{attribute 'qualified_only'}
VAR_GLOBAL

	Par1 		:BOOL:=TRUE;
	Par2		:INT:=10;
	Par3		:DINT:=100;
	Par4		:REAL:=100.1;
	Par5		:LREAL:=10.12;	

END_VAR

(* stored: Version 1.1.0.1, ProductVersion 3.1.4022.12
   GVL Merker: Id {4de0dba3-db52-482d-8e41-db9714b43ca4} *)
